// Mitsubishi GX Works2 project: P1_0724_ver01   PLC: Q03UDV

// global labels: Global1
VAR_GLOBAL
  그리퍼온솔 AT Y42 : BOOL;
  그리퍼오프솔 AT Y43 : BOOL;
  이송전진솔 AT Y40 : BOOL;
  이송후진솔 AT Y41 : BOOL;
  이송컨베이어 AT Y48 : BOOL;
  부품컨베이어 AT Y4F : BOOL;
  흡착패드 AT Y4E : BOOL;
  R_그리퍼온명령 AT X1000 : BOOL;
  R_그리퍼오프명령 AT X1001 : BOOL;
  R_흡착온명령 AT X1005 : BOOL;
  R_흡착오프명령 AT X1006 : BOOL;
  R_조립시작 AT X1007 : BOOL;
  R_이송완료 AT X1008 : BOOL;
  부품시작센서 AT X30 : BOOL;
  부품도착센서 AT X31 : BOOL;
  이송시작센서 AT X32 : BOOL;
  이송도착센서 AT X33 : BOOL;
  그리퍼온리드 AT X27 : BOOL;
  그리퍼오프리드 AT X28 : BOOL;
  TG1 AT X2A : BOOL;
  TG2 AT X2B : BOOL;
  TG3 AT X2C : BOOL;
  PB4 AT X2D : BOOL;
  PB5 AT X2E : BOOL;
  경광녹색 AT Y44 : BOOL;
  경광황색 AT Y45 : BOOL;
  경광적색 AT Y46 : BOOL;
  R그립온센서 AT Y1000 : BOOL;
  R그립오프센서 AT Y1001 : BOOL;
  R_로봇정지 AT X1009 : BOOL;
  R흡착온 AT Y1014 : BOOL;
  R흡착오프 AT Y1015 : BOOL;
  R부품도착 AT Y1016 : BOOL;
  R이송도착 AT Y1017 : BOOL;
  R이송시작 AT Y1018 : BOOL;
  R로봇시작 AT Y1019 : BOOL;
  R_재시작 AT Y1008 : BOOL;
  R_interrupt AT Y1009 : BOOL;
  부저 AT Y47 : BOOL;
  R이송중 AT Y1020 : BOOL;
END_VAR

PROGRAM MAIN
VAR
  그리퍼온 : BOOL;
  그리퍼오프 : BOOL;
  이송컨구동 : BOOL;
  흡착온 : BOOL;
  부품도착완료 : BOOL;
  T_흡착온대기 : TIMER;
  T_흡착오프대기 : TIMER;
  부품컨구동 : BOOL;
  T_부품감지대기 : TIMER;
  T_부품도착대기 : TIMER;
  이송시작 : BOOL;
  이송완료 : BOOL;
  T_부품에러 : TIMER;
  T_이송도착에러 : TIMER;
  에러발생 : BOOL;
  재시작 : BOOL;
  정지 : BOOL;
  이송배출 : BOOL;
  부품없음 : BOOL;
  T_이송에러 : TIMER;
END_VAR
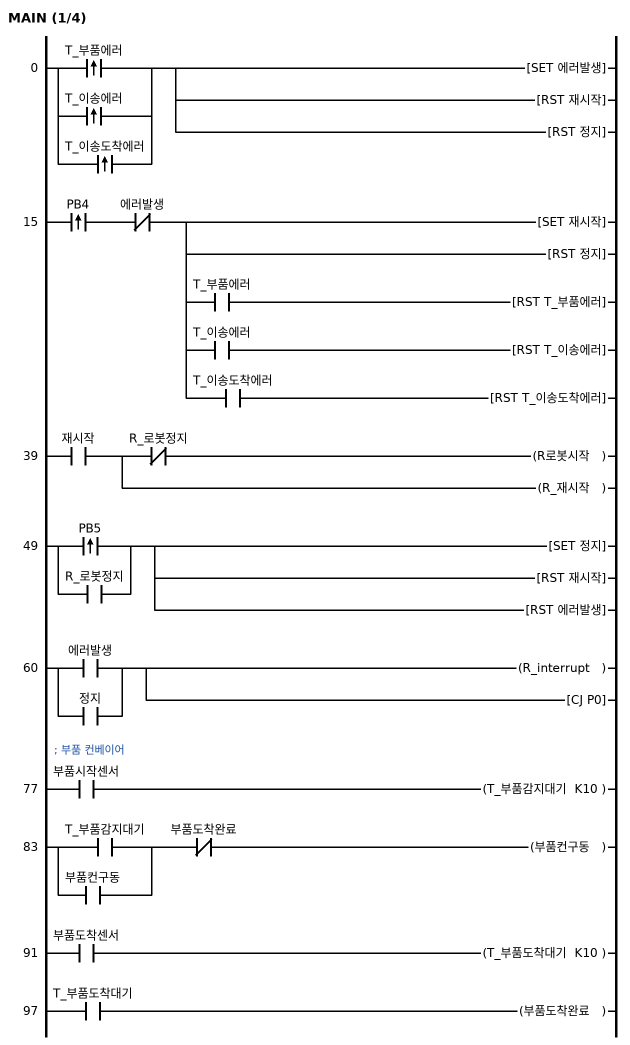
0     LDP     T_부품에러
      ORP     T_이송에러
      ORP     T_이송도착에러
      SET     에러발생
      RST     재시작
      RST     정지
15    LDP     PB4
      ANI     에러발생
      SET     재시작
      RST     정지
      MPS
      AND     T_부품에러
      RST     T_부품에러
      MRD
      AND     T_이송에러
      RST     T_이송에러
      MPP
      AND     T_이송도착에러
      RST     T_이송도착에러
39    LD      재시작
      MPS
      ANI     R_로봇정지
      OUT     R로봇시작
      MPP
      OUT     R_재시작
49    LDP     PB5
      OR      R_로봇정지
      SET     정지
      RST     재시작
      RST     에러발생
60    LD      에러발생
      OR      정지
      OUT     R_interrupt
      CJ      P0
; 부품 컨베이어
77    LD      부품시작센서
      OUT     T_부품감지대기 K10
83    LD      T_부품감지대기
      OR      부품컨구동
      ANI     부품도착완료
      OUT     부품컨구동
91    LD      부품도착센서
      OUT     T_부품도착대기 K10
97    LD      T_부품도착대기
      OUT     부품도착완료
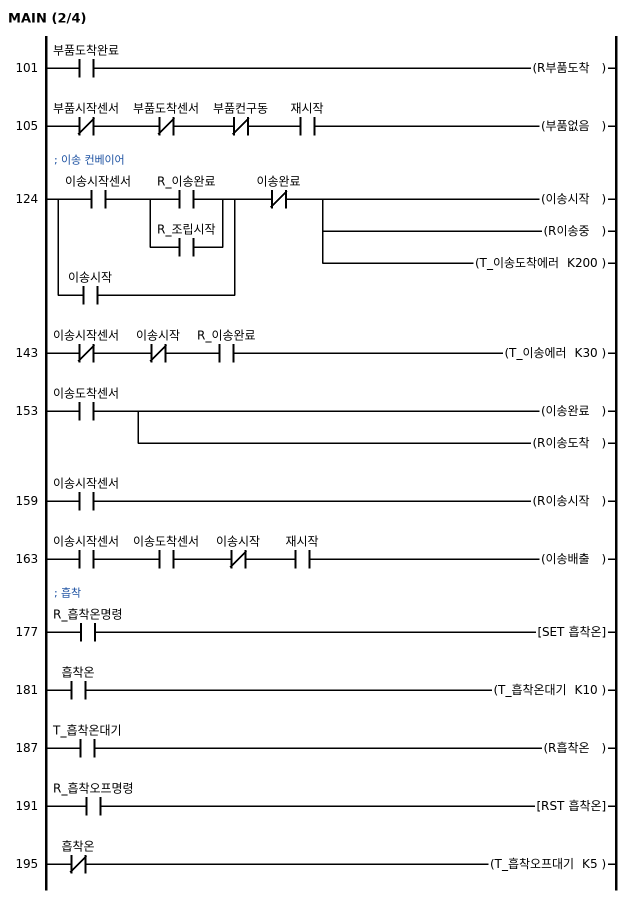
101   LD      부품도착완료
      OUT     R부품도착
105   LDI     부품시작센서
      ANI     부품도착센서
      ANI     부품컨구동
      AND     재시작
      OUT     부품없음
; 이송 컨베이어
124   LD      이송시작센서
      LD      R_이송완료
      OR      R_조립시작
      ANB
      OR      이송시작
      ANI     이송완료
      OUT     이송시작
      OUT     R이송중
      OUT     T_이송도착에러 K200
143   LDI     이송시작센서
      ANI     이송시작
      AND     R_이송완료
      OUT     T_이송에러 K30
153   LD      이송도착센서
      OUT     이송완료
      OUT     R이송도착
159   LD      이송시작센서
      OUT     R이송시작
163   LD      이송시작센서
      AND     이송도착센서
      ANI     이송시작
      AND     재시작
      OUT     이송배출
; 흡착
177   LD      R_흡착온명령
      SET     흡착온
181   LD      흡착온
      OUT     T_흡착온대기 K10
187   LD      T_흡착온대기
      OUT     R흡착온
191   LD      R_흡착오프명령
      RST     흡착온
195   LDI     흡착온
      OUT     T_흡착오프대기 K5
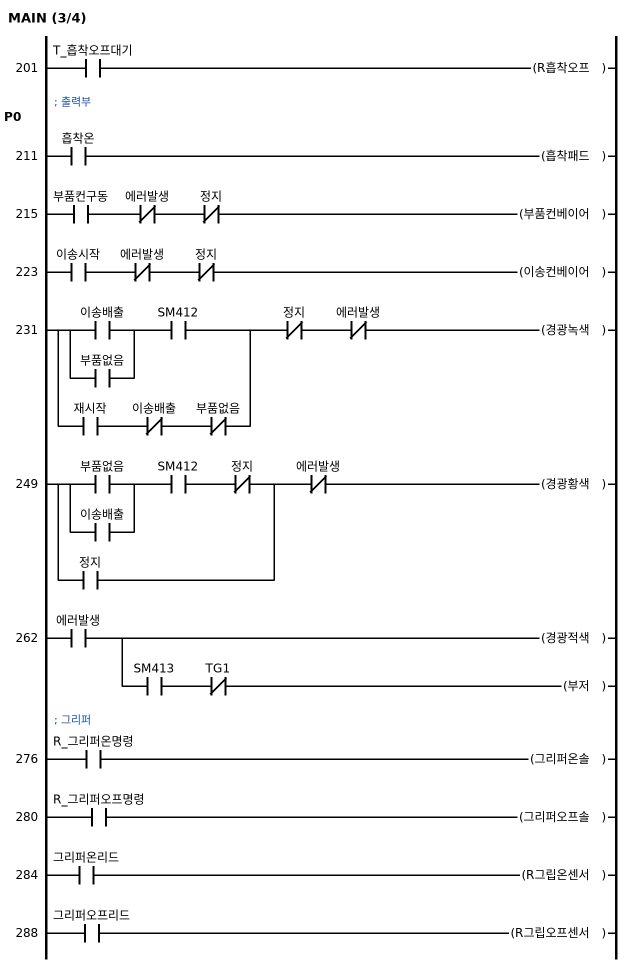
201   LD      T_흡착오프대기
      OUT     R흡착오프
; 출력부
      P0
211   LD      흡착온
      OUT     흡착패드
215   LD      부품컨구동
      ANI     에러발생
      ANI     정지
      OUT     부품컨베이어
223   LD      이송시작
      ANI     에러발생
      ANI     정지
      OUT     이송컨베이어
231   LD      이송배출
      OR      부품없음
      AND     SM412
      LD      재시작
      ANI     이송배출
      ANI     부품없음
      ORB
      ANI     정지
      ANI     에러발생
      OUT     경광녹색
249   LD      부품없음
      OR      이송배출
      AND     SM412
      ANI     정지
      OR      정지
      ANI     에러발생
      OUT     경광황색
262   LD      에러발생
      OUT     경광적색
      AND     SM413
      ANI     TG1
      OUT     부저
; 그리퍼
276   LD      R_그리퍼온명령
      OUT     그리퍼온솔
280   LD      R_그리퍼오프명령
      OUT     그리퍼오프솔
284   LD      그리퍼온리드
      OUT     R그립온센서
288   LD      그리퍼오프리드
      OUT     R그립오프센서
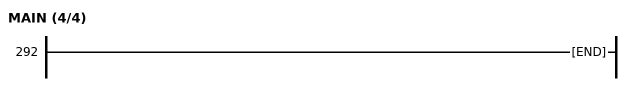
292   END
END_PROGRAM
